{attribute 'qualified_only'}
{attribute 'strict'}
TYPE L_Attenuators :
(
	AT1L0 := 1, // FEE Combo Gas/Solid Attenuator
    AT2L0 := 2 // FEE Solid Attenuator
);
END_TYPE

(* stored: Version 1.1.0.1, ProductVersion 3.1.4022.18
   EnumerationTextList L_Attenuators: Id {eed0cca7-59a7-44df-8ba0-3ca5777a6625} *)
